// TIA Portal V19 export
TYPE "SpeedMachine_CIn"
// stored: Access Published
   STRUCT
      Manager : "SpeedMachine_CIn_Manager";
      Bwd_ExtEnable : Bool := TRUE;
      Fwd_ExtEnable : Bool := TRUE;
      EnableManChangeVel : Bool := TRUE;   // Enable working of Manual velocity change Low to High
      ExternalPowerOn : Bool;
      ExternalAlarms : Bool := FALSE;
      VelocityOverride : Struct
         Enable : Bool := FALSE;
         Value : Real := 100.0;   // %
      END_STRUCT;
   END_STRUCT;
END_TYPE
